(* CODESYS project Fahrstuhl_Modell_Workspace.project

Project tree, tasks and I/O mapping:
  Device : CODESYS Control Win V3, 3S - Smart Software Solutions GmbH, order no. 305021, version 3.5.11.30
    application Application
      task DefaultTask (cyclic, interval T#10ms, priority 16) calls nothing
      Data types/
      Global Variables/
        global variables Globale_Variablen
      POUs/
      Visualizations/
        visualisation Fahrstuhl_Testbetrieb
        visualisation Fahrstuhl_Status
        visualisation Fahrstuhl_Bedienpult_Maschinenhaus
        visualisation Fahrstuhl_Bedienpult_Fahrkorb
        visualisation Fahrstuhl
        visualisation Doku1
      Symbols
      global variables PersistentVars
      trace Sampling_Trace (task ): 
  libraries: Standard, 3.5.9.0 (System)
  GlobalImagePool
  text list GlobalTextList
*)

// Device/Application/PersistentVars
VAR_GLOBAL PERSISTENT RETAIN
END_VAR

// Device/Application/Global Variables/Globale_Variablen
	VAR_GLOBAL


	Mot_Tuer_EGauf: BOOL;
	Mot_Tuer_EGzu: BOOL;
	Tuer_Auf_EG_ES: BOOL;  //Door opened fully
	Tuer_Zu_EG_ES: BOOL;   //Door closed fully
	// Light Baarier Sender
	Li_Tuer_EG: BOOL;
	Tuer_Si_EG: BOOL; // Light Barrier Receiver
	FK_VE_ue_EG: BOOL; // gnd Floor uPPER SWEEP POSITION
	FK_EL_EG: BOOL;  // gnd floor Middle Sweep position 
	FK_VE_un_EG: BOOL; //gnd floor Lowest Sweep position
	Anz_Ruf_EGauf: BOOL;
	In_Anford_EG:BOOL;  //gROUND FLOOR BUTTON
	Anf_EG_FK_Auf: BOOL; //Go uP BUTTON
	Tuer_Auf_EG:BOOL; //Door open ground floor (cONTROL PANEL)
	Tuer_Zu_EG:BOOL;
	Anz_Tuer_EG_Auf:BOOL;
	Anz_Tuer_EG_Zu:BOOL;
	Anz_FK_EG:BOOL;

	Mot_Tuer_1OGauf: BOOL;
	Mot_Tuer_1OGzu: BOOL;
	Tuer_Auf_1OG_ES: BOOL;
	Tuer_Zu_1OG_ES: BOOL;
	// Light Barrier Sender
	Li_Tuer_1OG: BOOL;
	Tuer_Si_1OG: BOOL;  // Light barrier receiver
	FK_VE_ue_1OG: BOOL;   //first Floor uPPER SWEEP POSITION
	FK_EL_1OG: BOOL;       // 1st floor Middle Sweep position 
	FK_VE_un_1OG: BOOL;     //1st floor Lowest Sweep position
	Anz_Ruf_1OGauf: BOOL;
	Anz_Ruf_1OGab: BOOL;
	Anz_1OG_Auf:BOOL;
	Anz_1OG_Ab:BOOL;
	In_Anford_1OG:BOOL;  //fIRST FLOOR BUTTON
	Anf_1OG_FK_Auf: BOOL; //Go uP BUTTON
	Anf_1OG_FK_Ab: BOOL;  //Go down button
	Tuer_Auf_1OG:BOOL;     //dOOr open 1st floor
	Tuer_Zu_1OG:BOOL;       //door closed 1st floor
	Anz_Tuer_1OG_Auf:BOOL;
	Anz_Tuer_1OG_Zu:BOOL;
	Anz_FK_1OG:BOOL;

	Mot_Tuer_2OGauf: BOOL;//
	Mot_Tuer_2OGzu: BOOL;
	Tuer_Auf_2OG_ES: BOOL;
	Tuer_Zu_2OG_ES: BOOL;
	// Light Barrier Sender
	Li_Tuer_2OG: BOOL;
	Tuer_Si_2OG: BOOL; // Light Barrier Receiver
	FK_VE_ue_2OG: BOOL;   //2nd Floor uPPER SWEEP POSITION
	FK_EL_2OG: BOOL;       // 2nd floor Middle Sweep position 
	FK_VE_un_2OG: BOOL;     //2nd floor Lowest Sweep position
	Anz_Ruf_2OGauf: BOOL;
	Anz_Ruf_2OGab: BOOL;
	Anz_2OG_Auf:BOOL;
	Anz_2OG_Ab:BOOL;
	In_Anford_2OG:BOOL;   //2ND FLOOR BUTTON
	Anf_2OG_FK_Auf: BOOL;   //Go uP BUTTON
	Anf_2OG_FK_Ab: BOOL;     //Go down BUTTON
	Tuer_Auf_2OG:BOOL;        //door open 2nd floor
	Tuer_Zu_2OG:BOOL;         //door closed 2nd floor
	Anz_Tuer_2OG_Auf:BOOL;
	Anz_Tuer_2OG_Zu:BOOL;
	Anz_FK_2OG:BOOL;

	Mot_Tuer_3OGauf: BOOL;
	Mot_Tuer_3OGzu: BOOL;
	Mot_Tuer_zu_3OG_man_sim: BOOL;
	Tuer_Auf_3OG_ES: BOOL; //Door opened fully
	Tuer_Zu_3OG_ES: BOOL; //Door closed fully
	// Light Barrier Sender
	Li_Tuer_3OG: BOOL;
	Tuer_Si_3OG: BOOL;  // Light barrier receiver
	FK_VE_ue_3OG: BOOL;   //3rd Floor uPPER SWEEP POSITION
	FK_EL_3OG: BOOL;       // 3rd floor Middle Sweep position
	FK_VE_un_3OG: BOOL;    //3rd floor Lowest Sweep position
	Anz_Ruf_3OGab: BOOL;
	In_Anford_3OG:BOOL;   //3RD FLOOR BUTTON
	Anf_3OG_FK_Ab: BOOL;  //Go uP down
	Tuer_Auf_3OG:BOOL;    //door open 3rd floor
	Tuer_Zu_3OG:BOOL;      //door closed 3rd floor    
	Anz_Tuer_3OG_Auf:BOOL;
	Anz_Tuer_3OG_Zu:BOOL;
	Anz_FK_3OG:BOOL;


	Mot_FK_Auf: BOOL;
	Mot_FK_Ab: BOOL;
	Fahrk_Auf:BOOL; //Car Open
	Fahrk_Ab:BOOL;  //CAR CLOSE
	Ue_Last:BOOL;  //Car Overload
	Anz_FK_Auf:BOOL;
	Anz_FK_Ab:BOOL;
	Anz_FK_zuhoch:BOOL;
	Anz_FK_zutief:BOOL;

	Tuer_Auf:BOOL; //Open the door
	NOTRUF: BOOL; //Emergency Csll
	IN_Steu_Ein: BOOL;  //Interior Controls
	Not_Aus:BOOL:=TRUE; //Emergency Stop Switch
	Betr_Art_Prog:BOOL;
	Anz_Prog:BOOL;
	Anz_Insp:BOOL;
	Anz_InnenST:BOOL;
	Anz_NOT_AUS_BP:BOOL;
	Anz_NOT_AUS_FK:BOOL;
	Lamp_Test:BOOL;
	Anf_Rel: BOOL;



	//INT_Bewegung_Stockwerke: INTEGRAL;
	Bewegung_Stockwerke_Visu: REAL;
	Bewegung_Stockwerke_inv:REAL;

	PROG:BOOL;
	Betriebsart:BOOL:=TRUE;  // program operation /Start
	PROG_Visu:BOOL;

	Hindernis_EG_sim: BOOL; //obstacle at gnd floor
	Hindernis_1OG_sim: BOOL; //obstacle at first floot
	Hindernis_2OG_sim: BOOL; //obstacle at 2nd floor
	Hindernis_3OG_sim: BOOL;  //obstacle at 3rd floor

END_VAR

// Device/Application/Visualizations/Fahrstuhl_Testbetrieb
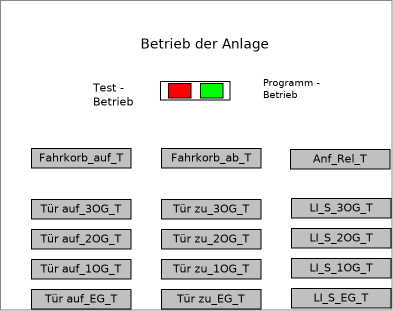
VISUALIZATION Fahrstuhl_Testbetrieb  // 393x311
    Rectangle (120,34 170x20), "Betrieb der Anlage"
    Rectangle (31,148 100x20), "Fahrkorb_auf_T", colour toggle: Visu_Fahrstuhl_Stockwerke.Motor_Fahrkorb_auf_T
        tap Visu_Fahrstuhl_Stockwerke.Motor_Fahrkorb_auf_T
    Rectangle (161,148 100x20), "Fahrkorb_ab_T", colour toggle: Visu_Fahrstuhl_Stockwerke.Motor_Fahrkorb_ab_T
        tap Visu_Fahrstuhl_Stockwerke.Motor_Fahrkorb_ab_T
    Rectangle (31,289 100x20), "Tür auf_EG_T", colour toggle: Visu_Fahrstuhl_Tueren.Mot_Tuer_auf_EG_T
        tap Visu_Fahrstuhl_Tueren.Mot_Tuer_auf_EG_T
    Rectangle (161,289 100x20), "Tür zu_EG_T", colour toggle: Visu_Fahrstuhl_Tueren.Mot_Tuer_zu_EG_T
        tap Visu_Fahrstuhl_Tueren.Mot_Tuer_zu_EG_T
    Rectangle (31,259 100x20), "Tür auf_1OG_T", colour toggle: Visu_Fahrstuhl_Tueren.Mot_Tuer_auf_1OG_T
        tap Visu_Fahrstuhl_Tueren.Mot_Tuer_auf_1OG_T
    Rectangle (161,259 100x20), "Tür zu_1OG_T", colour toggle: Visu_Fahrstuhl_Tueren.Mot_Tuer_zu_1OG_T
        tap Visu_Fahrstuhl_Tueren.Mot_Tuer_zu_1OG_T
    Rectangle (31,229 100x20), "Tür auf_2OG_T", colour toggle: Visu_Fahrstuhl_Tueren.Mot_Tuer_auf_2OG_T
        tap Visu_Fahrstuhl_Tueren.Mot_Tuer_auf_2OG_T
    Rectangle (161,229 100x20), "Tür zu_2OG_T", colour toggle: Visu_Fahrstuhl_Tueren.Mot_Tuer_zu_2OG_T
        tap Visu_Fahrstuhl_Tueren.Mot_Tuer_zu_2OG_T
    Rectangle (31,199 100x20), "Tür auf_3OG_T", colour toggle: Visu_Fahrstuhl_Tueren.Mot_Tuer_auf_3OG_T
        tap Visu_Fahrstuhl_Tueren.Mot_Tuer_auf_3OG_T
    Rectangle (161,199 100x20), "Tür zu_3OG_T", colour toggle: Visu_Fahrstuhl_Tueren.Mot_Tuer_zu_3OG_T
        tap Visu_Fahrstuhl_Tueren.Mot_Tuer_zu_3OG_T
    Rectangle (291,288 100x20), "LI_S_EG_T", colour toggle: Visu_Fahrstuhl_Tueren.Lischr_S_EG_T
        toggle Visu_Fahrstuhl_Tueren.Lischr_S_EG_T
    Rectangle (291,258 100x20), "LI_S_1OG_T", colour toggle: Visu_Fahrstuhl_Tueren.Lischr_S_1OG_T
        toggle Visu_Fahrstuhl_Tueren.Lischr_S_1OG_T
    Rectangle (291,228 100x20), "LI_S_2OG_T", colour toggle: Visu_Fahrstuhl_Tueren.Lischr_S_2OG_T
        toggle Visu_Fahrstuhl_Tueren.Lischr_S_2OG_T
    Rectangle (291,198 100x20), "LI_S_3OG_T", colour toggle: Visu_Fahrstuhl_Tueren.Lischr_S_3OG_T
        toggle Visu_Fahrstuhl_Tueren.Lischr_S_3OG_T
    Rectangle (160,81 70x19), invisible if: Globale_Variablen.PROG
        toggle Globale_Variablen.Betriebsart
    Rectangle (290,149 100x20), "Anf_Rel_T", colour toggle: Visu_Fahrstuhl_Stockwerke.Anf_Rel_T
        toggle Visu_Fahrstuhl_Stockwerke.Anf_Rel_T
    Rectangle (90,80 60x40), "Test - Betrieb"
    Rectangle (260,76 60x40), "Programm - Betrieb"
    Rectangle (168,83 23x15), invisible if: Globale_Variablen.Betriebsart
    Rectangle (200,83 23x15), invisible if: NOT Globale_Variablen.Betriebsart
END_VISUALIZATION

// Device/Application/Visualizations/Fahrstuhl_Status
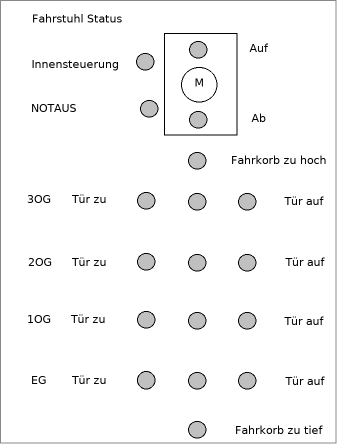
VISUALIZATION Fahrstuhl_Status  // 337x444
    Rectangle (164,33 73x102)
    Ellipse (181,67 36x35)
    Rectangle (188,72 23x22), "M"
    Ellipse (189,41 18x17), colour toggle: Globale_Variablen.Anz_FK_Auf
    Ellipse (140,100 18x17), colour toggle: Globale_Variablen.Anz_NOT_AUS_BP
    Ellipse (136,53 18x17), colour toggle: Globale_Variablen.Anz_InnenST
    Ellipse (188,421 18x17), colour toggle: Globale_Variablen.Anz_FK_zutief
    Ellipse (238,193 18x17), colour toggle: Globale_Variablen.Anz_Tuer_3OG_Auf
    Ellipse (137,192 18x17), colour toggle: Globale_Variablen.Anz_Tuer_3OG_Zu
    Ellipse (188,193 18x17), colour toggle: Globale_Variablen.Anz_FK_3OG
    Ellipse (188,152 18x17), colour toggle: Globale_Variablen.Anz_FK_zuhoch
    Ellipse (189,111 18x17), colour toggle: Globale_Variablen.Anz_FK_Ab
    Ellipse (238,254 18x17), colour toggle: Globale_Variablen.Anz_Tuer_2OG_Auf
    Ellipse (137,253 18x17), colour toggle: Globale_Variablen.Anz_Tuer_2OG_Zu
    Ellipse (188,254 18x17), colour toggle: Globale_Variablen.Anz_FK_2OG
    Ellipse (238,312 18x17), colour toggle: Globale_Variablen.Anz_Tuer_1OG_Auf
    Ellipse (137,311 18x17), colour toggle: Globale_Variablen.Anz_Tuer_1OG_Zu
    Ellipse (188,312 18x17), colour toggle: Globale_Variablen.Anz_FK_1OG
    Ellipse (238,372 18x17), colour toggle: Globale_Variablen.Anz_Tuer_EG_Auf
    Ellipse (137,371 18x18), colour toggle: Globale_Variablen.Anz_Tuer_EG_Zu
    Ellipse (188,372 18x17), colour toggle: Globale_Variablen.Anz_FK_EG
    Rectangle (27,53 97x23), "Innensteuerung"
    Rectangle (24,97 60x23), "NOTAUS"
    Rectangle (244,37 30x23), "Auf"
    Rectangle (244,107 30x23), "Ab"
    Rectangle (224,149 110x23), "Fahrkorb zu hoch"
    Rectangle (274,190 60x23), "Tür auf"
    Rectangle (275,251 60x23), "Tür auf"
    Rectangle (274,310 60x23), "Tür auf"
    Rectangle (275,370 60x23), "Tür auf"
    Rectangle (224,419 110x23), "Fahrkorb zu tief"
    Rectangle (65,188 49x23), "Tür zu"
    Rectangle (65,251 49x23), "Tür zu"
    Rectangle (64,308 49x23), "Tür zu"
    Rectangle (65,369 49x23), "Tür zu"
    Rectangle (24,188 30x23), "3OG"
    Rectangle (25,251 30x23), "2OG"
    Rectangle (24,308 30x23), "1OG"
    Rectangle (24,369 30x23), "EG"
    Rectangle (30,8 94x22), "Fahrstuhl Status"
END_VISUALIZATION

// Device/Application/Visualizations/Fahrstuhl_Bedienpult_Maschinenhaus
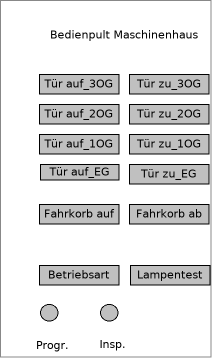
VISUALIZATION Fahrstuhl_Bedienpult_Maschinenhaus  // 212x358
    Rectangle (39,25 170x20), "Bedienpult Maschinenhaus"
    Rectangle (39,204 80x20), "Fahrkorb auf", colour toggle: Globale_Variablen.Fahrk_Auf
        tap Globale_Variablen.Fahrk_Auf
    Rectangle (129,204 80x20), "Fahrkorb ab", colour toggle: Globale_Variablen.Fahrk_Ab
        tap Globale_Variablen.Fahrk_Ab
    Rectangle (40,164 79x16), "Tür auf_EG", colour toggle: Globale_Variablen.Tuer_Auf_EG
        tap Globale_Variablen.Tuer_Auf_EG
    Rectangle (129,164 80x20), "Tür zu_EG", colour toggle: Globale_Variablen.Tuer_Zu_EG
        tap Globale_Variablen.Tuer_Zu_EG
    Rectangle (39,265 80x20), "Betriebsart", colour toggle: Globale_Variablen.Betr_Art_Prog
        toggle Globale_Variablen.Betr_Art_Prog
    Rectangle (39,134 80x20), "Tür auf_1OG", colour toggle: Globale_Variablen.Tuer_Auf_1OG
        tap Globale_Variablen.Tuer_Auf_1OG
    Rectangle (129,134 80x20), "Tür zu_1OG", colour toggle: Globale_Variablen.Tuer_Zu_1OG
        tap Globale_Variablen.Tuer_Zu_1OG
    Rectangle (39,104 80x20), "Tür auf_2OG", colour toggle: Globale_Variablen.Tuer_Auf_2OG
        tap Globale_Variablen.Tuer_Auf_2OG
    Rectangle (129,104 80x20), "Tür zu_2OG", colour toggle: Globale_Variablen.Tuer_Zu_2OG
        tap Globale_Variablen.Tuer_Zu_2OG
    Rectangle (39,74 80x20), "Tür auf_3OG", colour toggle: Globale_Variablen.Tuer_Auf_3OG
        tap Globale_Variablen.Tuer_Auf_3OG
    Rectangle (129,74 80x20), "Tür zu_3OG", colour toggle: Globale_Variablen.Tuer_Zu_3OG
        tap Globale_Variablen.Tuer_Zu_3OG
    Rectangle (130,265 80x20), "Lampentest", colour toggle: Globale_Variablen.Lamp_Test
        toggle Globale_Variablen.Lamp_Test
    Ellipse (40,304 18x17), colour toggle: Globale_Variablen.Anz_Prog
    Ellipse (100,304 18x17), colour toggle: Globale_Variablen.Anz_Insp
    Rectangle (30,335 45x21), "Progr."
    Rectangle (90,334 45x21), "Insp."
END_VISUALIZATION

// Device/Application/Visualizations/Fahrstuhl_Bedienpult_Fahrkorb
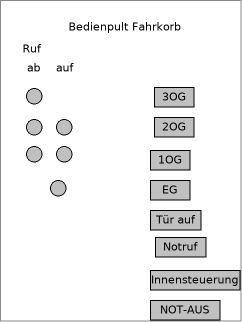
VISUALIZATION Fahrstuhl_Bedienpult_Fahrkorb  // 242x322
    Rectangle (65,17 120x20), "Bedienpult Fahrkorb"
    Rectangle (150,180 40x20), "EG", colour toggle: Globale_Variablen.In_Anford_EG
        tap Globale_Variablen.In_Anford_EG
    Rectangle (154,87 40x20), "3OG", colour toggle: Globale_Variablen.In_Anford_3OG
        tap Globale_Variablen.In_Anford_3OG
    Rectangle (154,117 40x20), "2OG", colour toggle: Globale_Variablen.In_Anford_2OG
        tap Globale_Variablen.In_Anford_2OG
    Rectangle (150,150 40x20), "1OG", colour toggle: Globale_Variablen.In_Anford_1OG
        tap Globale_Variablen.In_Anford_1OG
    Rectangle (150,270 90x20), "Innensteuerung", colour toggle: Globale_Variablen.IN_Steu_Ein
        toggle Globale_Variablen.IN_Steu_Ein
    Rectangle (150,300 70x20), "NOT-AUS", colour toggle: Globale_Variablen.Not_Aus
        toggle Globale_Variablen.Not_Aus
    Ellipse (26,88 16x16), colour toggle: Globale_Variablen.Anz_Ruf_3OGab
    Rectangle (150,210 51x20), "Tür auf", colour toggle: Globale_Variablen.Tuer_Auf
        tap Globale_Variablen.Tuer_Auf
    Rectangle (155,237 51x20), "Notruf", colour toggle: Globale_Variablen.NOTRUF
        tap Globale_Variablen.NOTRUF
    Ellipse (56,119 16x16), colour toggle: Globale_Variablen.Anz_Ruf_2OGauf
    Ellipse (26,119 16x16), colour toggle: Globale_Variablen.Anz_Ruf_2OGab
    Ellipse (56,146 16x16), colour toggle: Globale_Variablen.Anz_Ruf_1OGauf
    Ellipse (26,146 16x16), colour toggle: Globale_Variablen.Anz_Ruf_1OGab
    Ellipse (50,180 16x16), colour toggle: Globale_Variablen.Anz_Ruf_EGauf
    Rectangle (14,37 36x24), "Ruf"
    Rectangle (48,57 34x22), "auf"
    Rectangle (17,57 34x22), "ab"
END_VISUALIZATION

// Device/Application/Visualizations/Fahrstuhl
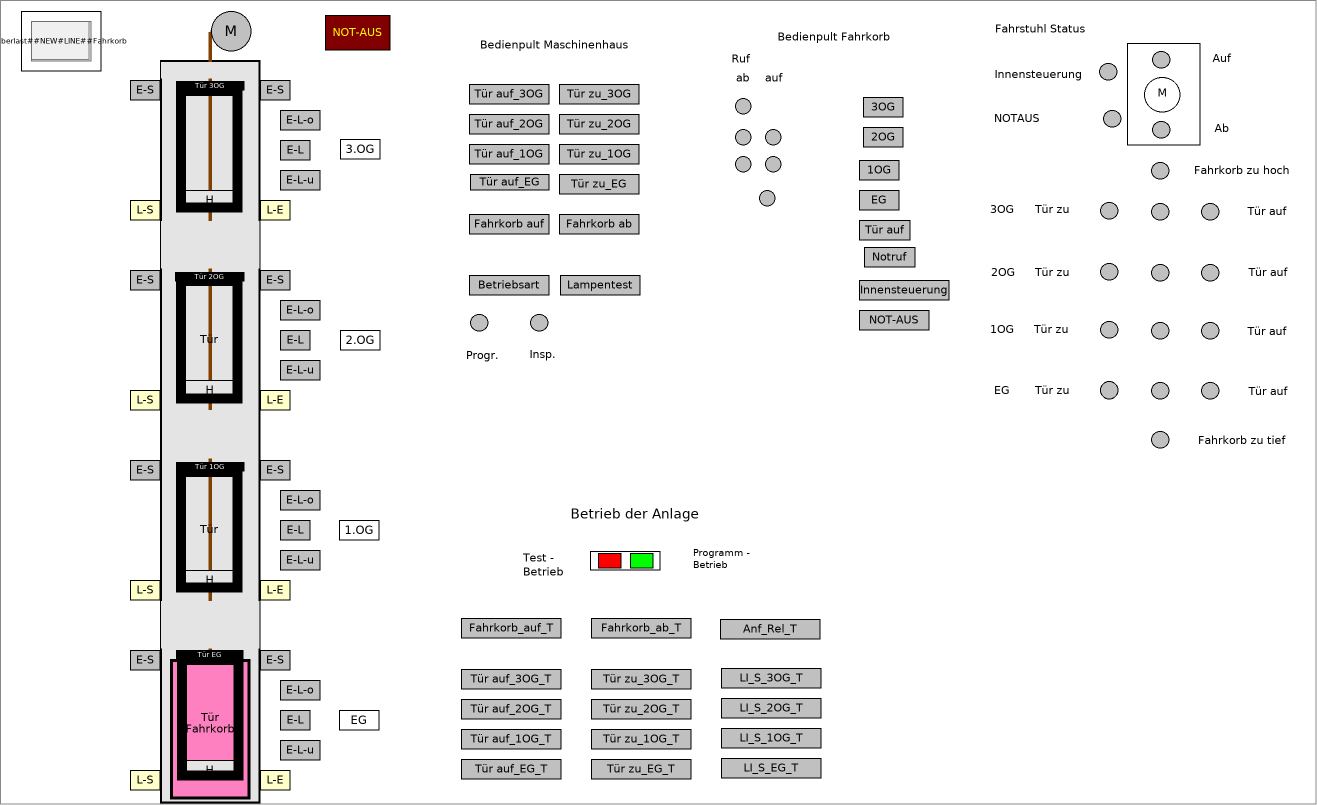
VISUALIZATION Fahrstuhl  // 1317x805
    Rectangle (160,60 100x743)
    Polygon (214,725), invisible if: NOT Visu_Fahrstuhl_Stockwerke.FK_unsichtbar
    Polygon (178,785), invisible if: NOT Visu_Fahrstuhl_Stockwerke.FK_unsichtbar
    Polygon (392,783), invisible if: NOT Visu_Fahrstuhl_Tueren.Tuer_EG_aus_Visu
    Polygon (392,594), invisible if: NOT Visu_Fahrstuhl_Tueren.Tuer_1OG_aus_Visu
    Polygon (392,405), invisible if: NOT Visu_Fahrstuhl_Tueren.Tuer_2OG_aus_Visu
    Polygon (392,214), invisible if: NOT Visu_Fahrstuhl_Tueren.Tuer_3OG_aus_Visu
    Rectangle (210,30 0x630), invisible if: Visu_Fahrstuhl_Stockwerke.FK_unsichtbar
        p1126004900: Globale_Variablen.Bewegung_Stockwerke_inv
    Rectangle (170,659 80x140), "Fahrkorb", invisible if: Visu_Fahrstuhl_Stockwerke.FK_unsichtbar
        p2773130477: Globale_Variablen.Bewegung_Stockwerke_inv
        p1126004900: Globale_Variablen.Bewegung_Stockwerke_inv
    Rectangle (161,601 98x47)
    Rectangle (162,410 95x48)
    Rectangle (161,221 98x47)
    Rectangle (161,62 97x16)
    Rectangle (180,760 60x20), "H", colour toggle: Globale_Variablen.Hindernis_EG_sim
        toggle Globale_Variablen.Hindernis_EG_sim
    Rectangle (180,190 60x20), "H", colour toggle: Globale_Variablen.Hindernis_3OG_sim
        toggle Globale_Variablen.Hindernis_3OG_sim
    Rectangle (180,380 60x20), "H", colour toggle: Globale_Variablen.Hindernis_2OG_sim
        toggle Globale_Variablen.Hindernis_2OG_sim
    Rectangle (180,570 60x20), "H", colour toggle: Globale_Variablen.Hindernis_1OG_sim
        toggle Globale_Variablen.Hindernis_1OG_sim
    Ellipse (211,11 40x40), "M", colour toggle: Visu_Fahrstuhl_Stockwerke.Mot_Ein_Visu
    Rectangle (130,650 30x20), "E-S", colour toggle: Globale_Variablen.Tuer_Zu_EG_ES
    Rectangle (260,650 30x20), "E-S", colour toggle: Globale_Variablen.Tuer_Auf_EG_ES
    Rectangle (130,460 30x20), "E-S", colour toggle: Globale_Variablen.Tuer_Zu_1OG_ES
    Rectangle (260,460 30x20), "E-S", colour toggle: Globale_Variablen.Tuer_Auf_1OG_ES
    Polygon (130,720), colour toggle: Globale_Variablen.Anf_EG_FK_Auf
        tap Globale_Variablen.Anf_EG_FK_Auf
    Rectangle (130,270 30x20), "E-S", colour toggle: Globale_Variablen.Tuer_Zu_2OG_ES
    Rectangle (260,270 30x20), "E-S", colour toggle: Globale_Variablen.Tuer_Auf_2OG_ES
    Rectangle (130,80 30x20), "E-S", colour toggle: Globale_Variablen.Tuer_Zu_3OG_ES
    Rectangle (260,80 30x20), "E-S", colour toggle: Globale_Variablen.Tuer_Auf_3OG_ES
    Polygon (130,520), colour toggle: Globale_Variablen.Anf_1OG_FK_Auf
        tap Globale_Variablen.Anf_1OG_FK_Auf
    Polygon (130,550), colour toggle: Globale_Variablen.Anf_1OG_FK_Ab
        tap Globale_Variablen.Anf_1OG_FK_Ab
    Polygon (130,330), colour toggle: Globale_Variablen.Anf_2OG_FK_Auf
        tap Globale_Variablen.Anf_2OG_FK_Auf
    Polygon (130,360), colour toggle: Globale_Variablen.Anf_2OG_FK_Ab
        tap Globale_Variablen.Anf_2OG_FK_Ab
    Polygon (130,170), colour toggle: Globale_Variablen.Anf_3OG_FK_Ab
        tap Globale_Variablen.Anf_3OG_FK_Ab
    Rectangle (339,710 40x20), "EG"
    Rectangle (340,139 40x20), "3.OG"
    Rectangle (340,330 40x20), "2.OG"
    Rectangle (339,520 40x20), "1.OG"
    Rectangle (280,680 40x20), "E-L-o", colour toggle: Globale_Variablen.FK_VE_ue_EG
    Rectangle (280,710 30x20), "E-L", colour toggle: Globale_Variablen.FK_EL_EG
    Rectangle (280,740 40x20), "E-L-u", colour toggle: Globale_Variablen.FK_VE_un_EG
    Rectangle (280,490 40x20), "E-L-o", colour toggle: Globale_Variablen.FK_VE_ue_1OG
    Rectangle (280,520 30x20), "E-L", colour toggle: Globale_Variablen.FK_EL_1OG
    Rectangle (280,550 40x20), "E-L-u", colour toggle: Globale_Variablen.FK_VE_un_1OG
    Rectangle (280,360 40x20), "E-L-u", colour toggle: Globale_Variablen.FK_VE_un_2OG
    Rectangle (280,330 30x20), "E-L", colour toggle: Globale_Variablen.FK_EL_2OG
    Rectangle (280,300 40x20), "E-L-o", colour toggle: Globale_Variablen.FK_VE_ue_2OG
    Rectangle (280,170 40x20), "E-L-u", colour toggle: Globale_Variablen.FK_VE_un_3OG
    Rectangle (280,140 30x20), "E-L", colour toggle: Globale_Variablen.FK_EL_3OG
    Rectangle (280,110 40x20), "E-L-o", colour toggle: Globale_Variablen.FK_VE_ue_3OG
    Rectangle (130,770 30x20), "L-S", colour toggle: Visu_Fahrstuhl_Tueren.Lischr_S_EG_Visu
    Polyline (170,220)
    Polyline (170,410)
    Polyline (170,600)
    Polyline (171,788)
    Polyline (360,220)
    Polyline (370,410)
    Polyline (370,600)
    Polyline (370,790)
    Polyline (230,10)
        p2858320360: Globale_Variablen.Bewegung_Stockwerke_Visu
    Polyline (250,30)
        p2858320360: Globale_Variablen.Bewegung_Stockwerke_Visu
    Rectangle (260,770 30x20), "L-E", colour toggle: Globale_Variablen.Tuer_Si_EG
    Rectangle (130,580 30x20), "L-S", colour toggle: Visu_Fahrstuhl_Tueren.Lischr_S_1OG_Visu
    Rectangle (260,580 30x20), "L-E", colour toggle: Globale_Variablen.Tuer_Si_1OG
    Rectangle (130,390 30x20), "L-S", colour toggle: Visu_Fahrstuhl_Tueren.Lischr_S_2OG_Visu
    Rectangle (260,390 30x20), "L-E", colour toggle: Globale_Variablen.Tuer_Si_2OG
    Rectangle (130,200 30x20), "L-S", colour toggle: Visu_Fahrstuhl_Tueren.Lischr_S_3OG_Visu
    Rectangle (260,200 30x20), "L-E", colour toggle: Globale_Variablen.Tuer_Si_3OG
    Polygon (130,70), colour toggle: Globale_Variablen.Anz_Ruf_3OGab
    Polygon (130,630), colour toggle: Globale_Variablen.Anz_Ruf_EGauf
    Polygon (130,230), colour toggle: Globale_Variablen.Anz_Ruf_2OGauf
    Polygon (130,420), colour toggle: Globale_Variablen.Anz_Ruf_1OGauf
    Polygon (130,260), colour toggle: Globale_Variablen.Anz_Ruf_2OGab
    Polygon (130,450), colour toggle: Globale_Variablen.Anz_Ruf_1OGab
    Frame (430,470 520x320), invisible if: Globale_Variablen.PROG
        shows Fahrstuhl_Testbetrieb()
    Frame (430,10 255x400)
        shows Fahrstuhl_Bedienpult_Maschinenhaus()
    Frame (709,10 248x400)
        shows Fahrstuhl_Bedienpult_Fahrkorb()
    Frame (963,10 352x462)
        shows Fahrstuhl_Status()
    Polygon (210,630), colour toggle: Visu_Fahrstuhl_Tueren.Lischr_S_EG_Visu
    Rectangle (176,467 66x125), "Tür", invisible if: Visu_Fahrstuhl_Tueren.Tuer_1OG_aus_Visu
        p3560616238: Visu_Fahrstuhl_Tueren.Bewegung_Tuer_1OG.CV
    Polygon (210,450), colour toggle: Globale_Variablen.Anz_1OG_Ab
    Polygon (210,420), colour toggle: Globale_Variablen.Anz_1OG_Auf
    Rectangle (176,276 66x127), "Tür", invisible if: Visu_Fahrstuhl_Tueren.Tuer_2OG_aus_Visu
        p3560616238: Visu_Fahrstuhl_Tueren.Bewegung_Tuer_2OG.CV
    Polygon (210,260), colour toggle: Globale_Variablen.Anz_2OG_Ab
    Polygon (210,230), colour toggle: Globale_Variablen.Anz_2OG_Auf
    Rectangle (176,86 66x126), invisible if: Visu_Fahrstuhl_Tueren.Tuer_3OG_aus_Visu
        p3560616238: Visu_Fahrstuhl_Tueren.Bewegung_Tuer_3OG.CV
    Polygon (210,70), colour toggle: Globale_Variablen.Mot_FK_Ab
    Rectangle (177,655 66x125), "Tür", invisible if: Visu_Fahrstuhl_Tueren.Tuer_EG_aus_Visu
        p3560616238: Visu_Fahrstuhl_Tueren.Bewegung_Tuer_EG.CV
    Rectangle (176,650 67x9), "Tür EG", invisible if: Visu_Fahrstuhl_Tueren.Tuer_EG_aus_Visu
        p3560616238: Visu_Fahrstuhl_Tueren.Bewegung_Tuer_EG.CV
    Rectangle (176,462 68x9), "Tür 1OG", invisible if: Visu_Fahrstuhl_Tueren.Tuer_1OG_aus_Visu
        p3560616238: Visu_Fahrstuhl_Tueren.Bewegung_Tuer_1OG.CV
    Rectangle (175,272 69x9), "Tür 2OG", invisible if: Visu_Fahrstuhl_Tueren.Tuer_2OG_aus_Visu
        p3560616238: Visu_Fahrstuhl_Tueren.Bewegung_Tuer_2OG.CV
    Rectangle (176,81 68x9), "Tür 3OG", invisible if: Visu_Fahrstuhl_Tueren.Tuer_3OG_aus_Visu
        p3560616238: Visu_Fahrstuhl_Tueren.Bewegung_Tuer_3OG.CV
    Group (21,11 78x58), colour toggle: Globale_Variablen.Ue_Last
        toggle Globale_Variablen.Ue_Last
        Rectangle (0,0 80x60), colour toggle: Globale_Variablen.Ue_Last
        Button (10,10 60x40), "Überlast##NEW#LINE##Fahrkorb", pressed state: Globale_Variablen.Ue_Last
            toggle Globale_Variablen.Ue_Last
    Rectangle (325,15 65x35), "NOT-AUS", colour toggle: Globale_Variablen.Anz_NOT_AUS_FK
END_VISUALIZATION

// Device/Application/Visualizations/Doku1
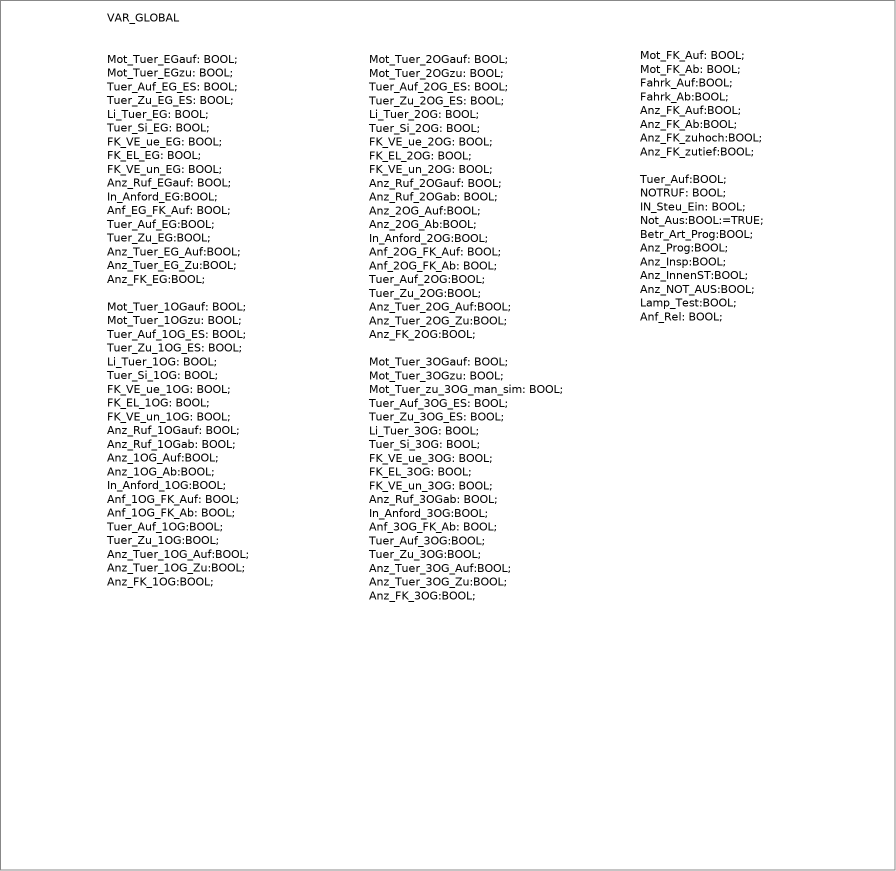
VISUALIZATION Doku1  // 896x871
    Rectangle (35,-28 324x871)
    Rectangle (97,10 224x841), "VAR_GLOBAL Mot_Tuer_EGauf: BOOL; Mot_Tuer_EGzu: BOOL; Tuer_Auf_EG_ES: BOOL; Tuer_Zu_EG_ES: BOOL; Li_Tuer_EG: BOOL; Tuer_Si_EG: BOOL; FK_VE_ue_EG: BOOL; FK_EL_EG: BOOL; FK_VE_un_EG: BOOL; Anz_Ruf_EGauf: BOOL; In_Anford_EG:BOOL; Anf_EG_FK_Auf: BOOL; Tuer_Auf_EG:BOOL; Tuer_Zu_EG:BOOL; Anz_Tuer_EG_Auf:BOOL; Anz_Tuer_EG_Zu:BOOL; Anz_FK_EG:BOOL; Mot_Tuer_1OGauf: BOOL; Mot_Tuer_1OGzu: BOOL; Tuer_Auf_1OG_ES: BOOL; Tuer_Zu_1OG_ES: BOOL; Li_Tuer_1OG: BOOL; Tuer_Si_1OG: BOOL; FK_VE_ue_1OG: BOOL; FK_EL_1OG: BOOL; FK_VE_un_1OG: BOOL; Anz_Ruf_1OGauf: BOOL; Anz_Ruf_1OGab: BOOL; Anz_1OG_Auf:BOOL; Anz_1OG_Ab:BOOL; In_Anford_1OG:BOOL; Anf_1OG_FK_Auf: BOOL; Anf_1OG_FK_Ab: BOOL; Tuer_Auf_1OG:BOOL; Tuer_Zu_1OG:BOOL; Anz_Tuer_1OG_Auf:BOOL; Anz_Tuer_1OG_Zu:BOOL; Anz_FK_1OG:BOOL;"
    Rectangle (359,24 264x845), "Mot_Tuer_2OGauf: BOOL; Mot_Tuer_2OGzu: BOOL; Tuer_Auf_2OG_ES: BOOL; Tuer_Zu_2OG_ES: BOOL; Li_Tuer_2OG: BOOL; Tuer_Si_2OG: BOOL; FK_VE_ue_2OG: BOOL; FK_EL_2OG: BOOL; FK_VE_un_2OG: BOOL; Anz_Ruf_2OGauf: BOOL; Anz_Ruf_2OGab: BOOL; Anz_2OG_Auf:BOOL; Anz_2OG_Ab:BOOL; In_Anford_2OG:BOOL; Anf_2OG_FK_Auf: BOOL; Anf_2OG_FK_Ab: BOOL; Tuer_Auf_2OG:BOOL; Tuer_Zu_2OG:BOOL; Anz_Tuer_2OG_Auf:BOOL; Anz_Tuer_2OG_Zu:BOOL; Anz_FK_2OG:BOOL; Mot_Tuer_3OGauf: BOOL; Mot_Tuer_3OGzu: BOOL; Mot_Tuer_zu_3OG_man_sim: BOOL; Tuer_Auf_3OG_ES: BOOL; Tuer_Zu_3OG_ES: BOOL; Li_Tuer_3OG: BOOL; Tuer_Si_3OG: BOOL; FK_VE_ue_3OG: BOOL; FK_EL_3OG: BOOL; FK_VE_un_3OG: BOOL; Anz_Ruf_3OGab: BOOL; In_Anford_3OG:BOOL; Anf_3OG_FK_Ab: BOOL; Tuer_Auf_3OG:BOOL; Tuer_Zu_3OG:BOOL; Anz_Tuer_3OG_Auf:BOOL; Anz_Tuer_3OG_Zu:BOOL; Anz_FK_3OG:BOOL;"
    Rectangle (630,20 264x843), "Mot_FK_Auf: BOOL; Mot_FK_Ab: BOOL; Fahrk_Auf:BOOL; Fahrk_Ab:BOOL; Anz_FK_Auf:BOOL; Anz_FK_Ab:BOOL; Anz_FK_zuhoch:BOOL; Anz_FK_zutief:BOOL; Tuer_Auf:BOOL; NOTRUF: BOOL; IN_Steu_Ein: BOOL; Not_Aus:BOOL:=TRUE; Betr_Art_Prog:BOOL; Anz_Prog:BOOL; Anz_Insp:BOOL; Anz_InnenST:BOOL; Anz_NOT_AUS:BOOL; Lamp_Test:BOOL; Anf_Rel: BOOL;"
    Rectangle (351,-18 485x27), "Globale Variablen die den virtuellen bzw. realen Fahrstuhl steuern."
END_VISUALIZATION
